// TwinCAT 3 PLC project TcUnit
// ProgramVersion: 3.1.4026.19
// libraries:
//   [AI Codes And Validation], * (Marden Edwards)
//   Tc2_Standard, * (Beckhoff Automation GmbH)
//   Tc2_System, * (Beckhoff Automation GmbH)
//   TcUnit, * (www.tcunit.org)
// project tree:
//   POUs/ PRG_TEST.TcPOU (not stored)
//   POUs/TcUnit/F_GetItemAITests/ F_GetItemAITests.TcPOU, PRG_GetItemAIManual.TcPOU
//   / TcUnit_Task.TcTTO (not stored)

// ---- POUs/TcUnit/F_GetItemAITests/F_GetItemAITests.TcPOU
FUNCTION_BLOCK F_GetItemAITests EXTENDS TcUnit.FB_TestSuite

VAR
	
	(* In/Out test*)		
	
END_VAR



//==============================================================
//01.CASE_Code
//==============================================================
Case_code01_GTIN_extractedWrong();
Case_code02_SERIAL_extractedWrong();
Case_code03_RSKU_extractedWrong();
Case_code04_BATCH_extractedWrong();
Case_code05_PO_extractedWrong();

//==============================================================
//02.Outer_Code
//==============================================================


//==============================================================
//03.Pack_Code
//==============================================================

METHOD INTERNAL Case_code01_GTIN_extractedWrong
VAR
	sFullCode		: T_MaxString;
	eCodeType		: CODE.E_CodeAI;
	stCodeInfo		: CODE.ST_CodeInfo;
	
	sF_GetItemAI	: T_MaxString;	
END_VAR
// Validation data init
stCodeInfo.eCodeType	:= CODE.E_CodeType.E_CASE;
TestInit(eCodeType := eCodeType, sFullCode := sFullcode, stCodeInfo := stCodeInfo);

//Change some data for test scenario below
sFullCode := '(01)17501031711052(21)86174He081137058500(240)10108245(10)86352024(91)5304012';
eCodeType	:= CODE.E_CodeAI.GTIN;


	
TcUnit.TEST('Case_code01_GTIN_extractedWrong');

	sF_GetItemAI := CODE.F_GetItemAI(sFullCode := sFullCode, 
									 eCodeType := eCodeType, 
									 stCodeInfo := stCodeInfo);
	
	AssertEquals_STRING(Expected:= '17501031711052', 
						Actual:= TO_STRING(sF_GetItemAI), 
						Message:= 'Wrong GTIN extracted');						

TEST_FINISHED();
END_METHOD

METHOD INTERNAL Case_code02_SERIAL_extractedWrong
VAR
	sFullCode		: T_MaxString;
	eCodeType		: CODE.E_CodeAI;
	stCodeInfo		: CODE.ST_CodeInfo;
	
	sF_GetItemAI	: T_MaxString;	
END_VAR
// Validation data init
stCodeInfo.eCodeType	:= CODE.E_CodeType.E_CASE;
TestInit(eCodeType := eCodeType, sFullCode := sFullcode, stCodeInfo := stCodeInfo);

//Change some data for test scenario below
sFullCode := '(01)17501031711052(21)86174He081137058500(240)10108245(10)86352024(91)5304012';
eCodeType	:= CODE.E_CodeAI.SERIAL;


	
TcUnit.TEST('Case_code02_SERIAL_extractedWrong');

	sF_GetItemAI := CODE.F_GetItemAI(sFullCode := sFullCode, 
									 eCodeType := eCodeType, 
									 stCodeInfo := stCodeInfo);
	
	AssertEquals_STRING(Expected:= '86174He081137058500', 
						Actual:= TO_STRING(sF_GetItemAI), 
						Message:= 'Wrong SERIAL extracted');						

TEST_FINISHED();
END_METHOD

METHOD INTERNAL Case_code03_RSKU_extractedWrong
VAR
	sFullCode		: T_MaxString;
	eCodeType		: CODE.E_CodeAI;
	stCodeInfo		: CODE.ST_CodeInfo;
	
	sF_GetItemAI	: T_MaxString;	
END_VAR
// Validation data init
stCodeInfo.eCodeType	:= CODE.E_CodeType.E_CASE;
TestInit(eCodeType := eCodeType, sFullCode := sFullcode, stCodeInfo := stCodeInfo);

//Change some data for test scenario below
sFullCode := '(01)17501031711052(21)86174He081137058500(240)10108245(10)86352024(91)5304012';
eCodeType	:= CODE.E_CodeAI.RSKU;


	
TcUnit.TEST('Case_code03_RSKU_extractedWrong');

	sF_GetItemAI := CODE.F_GetItemAI(sFullCode := sFullCode, 
									 eCodeType := eCodeType, 
									 stCodeInfo := stCodeInfo);
	
	AssertEquals_STRING(Expected:= '10108245', 
						Actual:= TO_STRING(sF_GetItemAI), 
						Message:= 'Wrong RSKU extracted');						

TEST_FINISHED();
END_METHOD

METHOD INTERNAL Case_code04_BATCH_extractedWrong
VAR
	sFullCode		: T_MaxString;
	eCodeType		: CODE.E_CodeAI;
	stCodeInfo		: CODE.ST_CodeInfo;
	
	sF_GetItemAI	: T_MaxString;	
END_VAR
// Validation data init
stCodeInfo.eCodeType	:= CODE.E_CodeType.E_CASE;
TestInit(eCodeType := eCodeType, sFullCode := sFullcode, stCodeInfo := stCodeInfo);

//Change some data for test scenario below
sFullCode := '(01)17501031711052(21)86174He081137058500(240)10108245(10)86352024(91)5304012';
eCodeType	:= CODE.E_CodeAI.BATCH;


	
TcUnit.TEST('Case_code04_BATCH_extractedWrong');

	sF_GetItemAI := CODE.F_GetItemAI(sFullCode := sFullCode, 
									 eCodeType := eCodeType, 
									 stCodeInfo := stCodeInfo);
	
	AssertEquals_STRING(Expected:= '86352024', 
						Actual:= TO_STRING(sF_GetItemAI), 
						Message:= 'Wrong BATCH extracted');						

TEST_FINISHED();
END_METHOD

METHOD INTERNAL Case_code05_PO_extractedWrong
VAR
	sFullCode		: T_MaxString;
	eCodeType		: CODE.E_CodeAI;
	stCodeInfo		: CODE.ST_CodeInfo;
	
	sF_GetItemAI	: T_MaxString;	
END_VAR
// Validation data init
stCodeInfo.eCodeType	:= CODE.E_CodeType.E_CASE;
TestInit(eCodeType := eCodeType, sFullCode := sFullcode, stCodeInfo := stCodeInfo);

//Change some data for test scenario below
sFullCode := '(01)17501031711052(21)86174He081137058500(240)10108245(10)86352024(91)5304012';
eCodeType	:= CODE.E_CodeAI.PO;


	
TcUnit.TEST('Case_code05_PO_extractedWrong');

	sF_GetItemAI := CODE.F_GetItemAI(sFullCode := sFullCode, 
									 eCodeType := eCodeType, 
									 stCodeInfo := stCodeInfo);
	
	AssertEquals_STRING(Expected:= '5304012', 
						Actual:= TO_STRING(sF_GetItemAI), 
						Message:= 'Wrong PO extracted');						

TEST_FINISHED();
END_METHOD

METHOD PRIVATE TestInit
VAR_IN_OUT
	eCodeType		: CODE.E_CodeAI;
	stCodeInfo		: CODE.ST_CodeInfo;
	sFullCode		: T_MaxString;
END_VAR

VAR	
END_VAR

// Case validation recipe
IF stCodeInfo.eCodeType = CODE.E_CodeType.E_CASE THEN

// GTIN 
	stCodeInfo.stGTIN.sStartAI := '(01)';
	stCodeInfo.stGTIN.sEndAI := '(';
	stCodeInfo.stGTIN.nCodeLength := 14;
	stCodeInfo.stGTIN.nCodeStartPos := 0;	
	
// SERIAL	
	stCodeInfo.stSerialCode.sStartAI := '(21)';
	stCodeInfo.stSerialCode.sEndAI := '(';
	stCodeInfo.stSerialCode.nCodeLength := 19;
	stCodeInfo.stSerialCode.nCodeStartPos := 0;	
	
// RSKU
	stCodeInfo.stRSKU.sStartAI := '(240)';
	stCodeInfo.stRSKU.sEndAI := '(';
	stCodeInfo.stRSKU.nCodeLength := 8;
	stCodeInfo.stRSKU.nCodeStartPos := 0;	
	
// BATCH
	stCodeInfo.stBatchID.sStartAI := '(10)';
	stCodeInfo.stBatchID.sEndAI := '(';
	stCodeInfo.stBatchID.nCodeLength := 8;
	stCodeInfo.stBatchID.nCodeStartPos := 0;	
	
// PRODUCTION ORDER
	stCodeInfo.stProductionOrder.sStartAI := '(91)';
	stCodeInfo.stProductionOrder.sEndAI := '(';
	stCodeInfo.stProductionOrder.nCodeLength := 7;
	stCodeInfo.stProductionOrder.nCodeStartPos := 0;	

stCodeInfo.nMinLength 		:= 10; // NOT used
stCodeInfo.nEntireLength	:= 77;
stCodeInfo.nNumberOfAIs		:= 5;
	
ELSIF stCodeInfo.eCodeType = CODE.E_CodeType.E_OUTER THEN
	;

ELSIF stCodeInfo.eCodeType = CODE.E_CodeType.E_PACK THEN
	;

END_IF
END_METHOD

END_FUNCTION_BLOCK

// ---- POUs/TcUnit/F_GetItemAITests/PRG_GetItemAIManual.TcPOU
PROGRAM PRG_GetItemAIManual
VAR
	sFullCode		: T_MaxString;
	eCodeType		: CODE.E_CodeAI;
	stCodeInfo		: CODE.ST_CodeInfo;
	
	sF_GetItemAI	: T_MaxString;

END_VAR

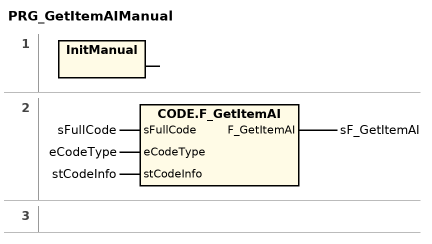
// NETWORK 1
InitManual();

// NETWORK 2
sF_GetItemAI := CODE.F_GetItemAI(sFullCode := sFullCode, eCodeType := eCodeType, stCodeInfo := stCodeInfo);

// NETWORK 3

ACTION InitManual:

sFullCode	:= '(01)17501031711052(21)86174He081137058500(240)10108245(10)86352024(91)5304012';
stCodeInfo.eCodeType	:= CODE.E_CodeType.E_CASE;

	
//eCodeType	:= CODE.E_CodeAI.GTIN;
eCodeType	:= CODE.E_CodeAI.SERIAL;
//eCodeType	:= CODE.E_CodeAI.RSKU;
//eCodeType	:= CODE.E_CodeAI.BATCH;
//eCodeType	:= CODE.E_CodeAI.PO;


// GTIN 
	stCodeInfo.stGTIN.sStartAI := '(01)';
	stCodeInfo.stGTIN.sEndAI := '(';
	stCodeInfo.stGTIN.nCodeLength := 14;
	stCodeInfo.stGTIN.nCodeStartPos := 0;	
	
// SERIAL	
	stCodeInfo.stSerialCode.sStartAI := '(21)';
	stCodeInfo.stSerialCode.sEndAI := '(';
	stCodeInfo.stSerialCode.nCodeLength := 19;
	stCodeInfo.stSerialCode.nCodeStartPos := 0;	
	
// RSKU
	stCodeInfo.stRSKU.sStartAI := '(240)';
	stCodeInfo.stRSKU.sEndAI := '(';
	stCodeInfo.stRSKU.nCodeLength := 8;
	stCodeInfo.stRSKU.nCodeStartPos := 0;	
	
// BATCH
	stCodeInfo.stBatchID.sStartAI := '(10)';
	stCodeInfo.stBatchID.sEndAI := '(';
	stCodeInfo.stBatchID.nCodeLength := 8;
	stCodeInfo.stBatchID.nCodeStartPos := 0;	
	
// PRODUCTION ORDER
	stCodeInfo.stProductionOrder.sStartAI := '(91)';
	stCodeInfo.stProductionOrder.sEndAI := '(';
	stCodeInfo.stProductionOrder.nCodeLength := 7;
	stCodeInfo.stProductionOrder.nCodeStartPos := 0;	



stCodeInfo.nMinLength 		:= 10;
stCodeInfo.nEntireLength	:= 77;
stCodeInfo.nNumberOfAIs		:= 5;
END_ACTION

END_PROGRAM
